{attribute 'qualified_only'}
VAR_GLOBAL
	Enc_Axis: AXIS_REF;
	Conveyor_Speed :	LREAL	;
	Encoder_Value	:	LREAL	;
	Real_Position: LREAL;
	Real_Velocity: LREAL;
	Count	AT%I*	:INT;
	Conveyor_CW AT%Q* : BOOL	;
	Conveyor_CCW AT%Q* : BOOL	;
	
END_VAR

(* stored: Version 1.1.0.1, ProductVersion 3.1.4024.15
   GVL GVL_Encoder: Id {89f3ab96-2606-45cb-b9c5-9fa7df819b12} *)
